(* CoDeSys 2.3.9.41 project: PLC2.pro *)
(* Libraries: STANDARD.LIB 4.10.05 11:14:46, IECSFC.LIB 13.4.06 15:51:28, SYSLIBTIME.LIB 6.11.19 15:29:28, ANALYZATION.LIB 5.10.99 09:05:06 *)

(* PLC configuration (modules and I/O channels)
Fast discrete inputs [I_SIMPLE_INPUT] node 0, in %IB0 out %QB0 {ChannellName = Fast discrete inputs; Filtrationtime = 10000}
  AT %IX0.0 [BitInput] Discrete input 1 {ChannellName = Enter name}
  AT %IX0.1 [BitInput] Discrete input 2 {ChannellName = Enter name}
  AT %IX0.2 [BitInput] Discrete input 3 {ChannellName = Enter name}
  AT %IX0.3 [BitInput] Discrete input 4 {ChannellName = Enter name}
Discrete inputs [ID130] node 1, in %IB1 out %QB1 {ChannellName = Discrete inputs; Filtrationtime_GeneralINP = 10; PinCount = 12; Visibility = No}
  AT %IB1.0 [ByteInput] 8 discrete inputs {ChannellName = Enter name}
  AT %IB1.1 [ByteInput] 4 discrete inputs {ChannellName = Enter name}
Fast discrete outputs [OWEN_ID570] node 2, in %IB2 out %QB2 {ChannellName = Fast discrete outputs; SafeValueBool = FALSE; SafeValueBool = FALSE; SafeValueBool = FALSE; SafeValueBool = FALSE; Visibility = No}
  DO1 AT %QX2.0 [BitOutput] Fast discrete output 1 {ChannellName = Enter name}
  DO2 AT %QX2.1 [BitOutput] Fast discrete output 2 {ChannellName = Enter name}
  DO3 AT %QX2.2 [BitOutput] Fast discrete output 3 {ChannellName = Enter name}
  AT %QX2.3 [BitOutput] Fast discrete output 4 {ChannellName = Enter name}
AT %QB3.0 [ByteOutput] 8 discrete outputs {ChannellName = Enter name}
AT %QB3.1 [ByteOutput] 8 discrete outputs {ChannellName = Enter name}
Fast analog inputs [ID125] node 4, in %IB4 out %QB4 {ChannellName = Fast analog inputs; Flt_Comm = 50Hz 2Por}
  AT %IR4.0 [FloatInputP] You need to reboot PLC after change AI configuration! {ChannellName = Fast analog input; AIN_TYPE = 4-20 mA; Peak_Filtr = 200; Flt_Ch = Off; TauRC = 10; MinFV = 0; MaxFV = 20000.0}
  AT %IR4.1 [FloatInputP] You need to reboot PLC after change AI configuration! {ChannellName = Fast analog input; AIN_TYPE = 4-20 mA; Peak_Filtr = 200; Flt_Ch = Off; TauRC = 10; MinFV = 0; MaxFV = 20000.0}
  AT %IR4.2 [FloatInputP] You need to reboot PLC after change AI configuration! {ChannellName = Fast analog input; AIN_TYPE = 4-20 mA; Peak_Filtr = 200; Flt_Ch = Off; TauRC = 10; MinFV = 0; MaxFV = 20000.0}
  AT %IR4.3 [FloatInputP] You need to reboot PLC after change AI configuration! {ChannellName = Fast analog input; AIN_TYPE = 4-20 mA; Peak_Filtr = 200; Flt_Ch = Off; TauRC = 10; MinFV = 0; MaxFV = 20000.0}
  AT %IR4.4 [FloatInputP] You need to reboot PLC after change AI configuration! {ChannellName = Fast analog input; AIN_TYPE = 4-20 mA; Peak_Filtr = 200; Flt_Ch = Off; TauRC = 10; MinFV = 0; MaxFV = 20000.0}
  AT %IR4.5 [FloatInputP] You need to reboot PLC after change AI configuration! {ChannellName = Fast analog input; AIN_TYPE = 4-20 mA; Peak_Filtr = 200; Flt_Ch = Off; TauRC = 10; MinFV = 0; MaxFV = 20000.0}
  AT %IR4.6 [FloatInputP] You need to reboot PLC after change AI configuration! {ChannellName = Fast analog input; AIN_TYPE = 4-20 mA; Peak_Filtr = 200; Flt_Ch = Off; TauRC = 10; MinFV = 0; MaxFV = 20000.0}
  AT %IR4.7 [FloatInputP] You need to reboot PLC after change AI configuration! {ChannellName = Fast analog input; AIN_TYPE = 4-20 mA; Peak_Filtr = 200; Flt_Ch = Off; TauRC = 10; MinFV = 0; MaxFV = 20000.0}
  AT %IW4.8 [WordInput] AI read time (10ms) {ChannellName = Enter name}
Analog outputs [ID126] node 5, in %IB5 out %QB5 {ChannellName = Analog outputs}
  AT %QR5.0 [FloatOutputP] AO #1 {ChannellName = Analog output; AOUT_TYPE = 4-20 mA; SafeValueREAL = 0.0}
  AT %QR5.1 [FloatOutputP] AO #2 {ChannellName = Analog output; AOUT_TYPE = 4-20 mA; SafeValueREAL = 0.0}
  AT %QR5.2 [FloatOutputP] AO #3 {ChannellName = Analog output; AOUT_TYPE = 4-20 mA; SafeValueREAL = 0.0}
  AT %QR5.3 [FloatOutputP] AO #4 {ChannellName = Analog output; AOUT_TYPE = 4-20 mA; SafeValueREAL = 0.0}
Special input [ID103] node 6, in %IB6 out %QB6 {ChannellName = Special input}
  AT %IX6.0 [BitInput] Special input {ChannellName = Enter name}
Special output [ID104] node 7, in %IB7 out %QB7 {ChannellName = Special output}
  AT %QX7.0 [BitOutput] Special output {ChannellName = Enter name}
ModBus (Master) [MODBUS_MASTER_ID450] node 8, in %IB8 out %QB8 {ChannellName = ModBus (Master); Visibility = No}
  AT %QD8.0 [DWordOutput] Last address {ChannellName = Enter name}
  AT %QW8.1 [WordOutput] Last error {ChannellName = Enter name}
  RS-485-1 [COM1_USART] node 0, in %IB8.0 out %QB8.0 {ChannellName = RS-485-1; CommunicationSpeed = 115200; Parity = NO PARITY CHECK; BitLength = 8 bits; StopLength = One stop bit; InterfaceType = RS485; FrameOriented = RTU; Timeout = 0; Visibility = No}
start1 AT %QB8.1.0 [ComChannel] Command (0xff - Start) {ChannellName = Enter name}
readTwoBytesFromPLC1_1 AT %QW8.1.0.0 [WordOutput] {ChannellName = Enter name}
start2 AT %QB8.2.0 [ComChannel] Command (0xff - Start) {ChannellName = Enter name}
readTwoBytesFromPLC1_2 AT %QW8.2.0.0 [WordOutput] {ChannellName = Enter name}
start3 AT %QB8.3.0 [ComChannel] Command (0xff - Start) {ChannellName = Enter name}
readTwoBytesFromPLC1_3 AT %QW8.3.0.0 [WordOutput] {ChannellName = Enter name}
TCP [TCP_ID221] node 0, in %IB9.0.0 out %QB9.0.0 {ChannellName = TCP; RemotePort = 502; Visibility = No}
float_1 AT %QD9.1.0 [FloatOutput] {ChannellName = Enter name}
uint_1 AT %QW9.2.0 [WordOutput] {ChannellName = Enter name}
*)

(* POU PLC_PRG, CFC *)
PROGRAM PLC_PRG
VAR
	boolStab: BOOL;
	rtrig: R_TRIG;
	init: BOOL;
	TON: TON;
	rtrig2: R_TRIG;
	rtrig3: R_TRIG;
END_VAR
VAR (* helpers for the ST form of the networks *)
	_t61 : BOOL;
END_VAR
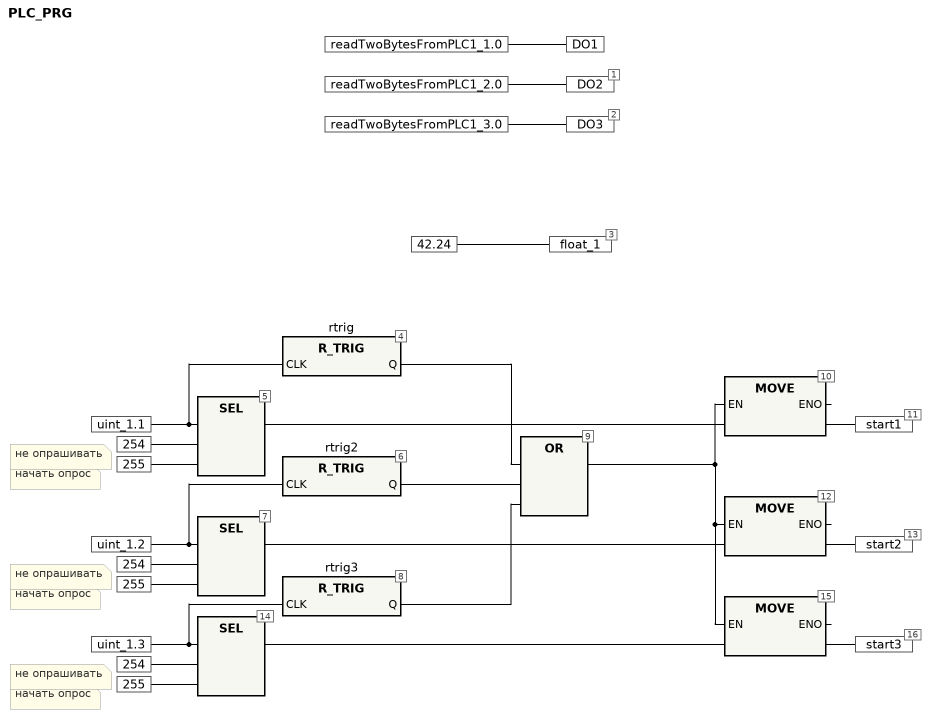
_CFC_ (* Continuous Function Chart, elements in execution order *)
(* начать опрос *)
(* не опрашивать *)
(* начать опрос *)
(* не опрашивать *)
(* начать опрос *)
(* не опрашивать *)
#0 DO1 <= readTwoBytesFromPLC1_1.0
#1 DO2 <= readTwoBytesFromPLC1_2.0
#2 DO3 <= readTwoBytesFromPLC1_3.0
#3 float_1 <= 42.24
#4 rtrig:R_TRIG(CLK: uint_1.1)
#5 SEL(uint_1.1, 254, 255)
#6 rtrig2:R_TRIG(CLK: uint_1.2)
#7 SEL(uint_1.2, 254, 255)
#8 rtrig3:R_TRIG(CLK: uint_1.3)
#9 OR(#4.Q, #6.Q, #8.Q)
#10 MOVE(EN: #9, #5)
#11 start1 <= #10
#12 MOVE(EN: #9, #7)
#13 start2 <= #12
#14 SEL(uint_1.3, 254, 255)
#15 MOVE(EN: #9, #14)
#16 start3 <= #15
_END_CFC_
(* the same logic as Structured Text *)
(* начать опрос *)
(* не опрашивать *)
(* начать опрос *)
(* не опрашивать *)
(* начать опрос *)
(* не опрашивать *)
DO1 := readTwoBytesFromPLC1_1.0;
DO2 := readTwoBytesFromPLC1_2.0;
DO3 := readTwoBytesFromPLC1_3.0;
float_1 := 42.24;
rtrig(CLK := uint_1.1);
rtrig2(CLK := uint_1.2);
rtrig3(CLK := uint_1.3);
_t61 := rtrig.Q OR rtrig2.Q OR rtrig3.Q;
IF _t61 THEN start1 := SEL(uint_1.1, 254, 255); END_IF;
IF _t61 THEN start2 := SEL(uint_1.2, 254, 255); END_IF;
IF _t61 THEN start3 := SEL(uint_1.3, 254, 255); END_IF;
END_PROGRAM
